FUNCTION_BLOCK FB_BiDirectionConveyor EXTENDS FB_Conveyor
VAR_INPUT
    bSensorAisleEntry   : BOOL;    // Physical Sensor at the Loop Junction
END_VAR

VAR_OUTPUT
    bMotorReverse       : BOOL;    // Physical Output for Reverse direction
END_VAR

VAR
    // No new internal timers needed yet, as we reuse the Parent's JamTimer
END_VAR

// 1. Run the Parent Logic (Handles Enable, Reset, and Forward Jamming)
SUPER^();

// 2. Specific Logic for Reverse/Waiting states
CASE eConveyorMode OF
    
    E_ConveyorMode.IDLE:
        bMotorReverse := FALSE;
        // bMotorRun is already handled by the Parent IDLE state

    E_ConveyorMode.TRANSPORT_TO_LOOP:
        bMotorRun     := TRUE;   // Turn on power
        bMotorReverse := TRUE;   // Set direction to Reverse
        
        // Transition: Stop when the box reaches the Loop junction sensor
        IF bSensorAisleEntry THEN
            eConveyorMode := E_ConveyorMode.WAITING_FOR_LOOP;
        END_IF

    E_ConveyorMode.WAITING_FOR_LOOP:
        bMotorRun     := FALSE;
        bMotorReverse := FALSE;

    E_ConveyorMode.FAULT:
        bMotorReverse := FALSE;
        // bMotorRun is already set to FALSE by the Parent FAULT state

END_CASE

METHOD M_Run : BOOL
VAR_INPUT
	bForward : BOOL;
END_VAR

// Only allow starting if not in Fault
IF eConveyorMode <> E_ConveyorMode.FAULT AND bEnable THEN
    
    IF bForward THEN
        eConveyorMode := E_ConveyorMode.TRANSPORT_TO_CRANE;
    ELSE
        eConveyorMode := E_ConveyorMode.TRANSPORT_TO_LOOP;
    END_IF
    
    M_Run := TRUE;
ELSE
    M_Run := FALSE;
END_IF
END_METHOD

END_FUNCTION_BLOCK

(* stored: Version 1.1.0.1, ProductVersion 3.1.4024.16
   POU FB_BiDirectionConveyor: Id {82de352f-fae1-461d-8e99-3962df4892ff}, SpecialFunc None
   Method M_Run: Id {9fa79b56-5384-4ec4-a8a5-f6e5246fc03d} *)
